PROGRAM MAIN
VAR
END_VAR

END_PROGRAM

(* stored: Version 1.1.0.1
   POU MAIN: Id {6c4c3d1f-c9cd-4279-8e17-c067dff067d5} *)
